// TIA Portal V20 export
DATA_BLOCK "ControlNodes"   // DB72
// stored: MemoryReserve 100, Namespace Unit1.Em7
   VAR
      em : "LAF_typeEmControlNode";
      emstate { S7_SetPoint := 'True'} : "LUC_typeStates";
      cm : "Unit1.Em7.typeCmControlNode";
      citiMap : Struct
         PMC : "LER_PMC_Input_Data";
         FlexNet { S7_SetPoint := 'True'} : "LER_FlexNet_Data";
      END_STRUCT;
      hotPressRight : "Unit1.Em7.typeSequenceControlNode";
      emData : "Unit1.Em7.typeEmDataControlNode";
      SpecialFunctionMode : Struct
         DryRun : Struct
            JRdetectPV : Array[0..15] of Bool;
         END_STRUCT;
      END_STRUCT;
      cmHotPressRightSafetyPin : "LBC_typeDigitalSignalControlNode";
      cmHotPressRightJRDetect : "LBC_typeDigitalSignalControlNode";
      cmHotPressRightStageLiftFrontUpDown : "LBC_typeTwoWayActuatorControlNode";
      cmHotPressRightStageLiftRearUpDown : "LBC_typeTwoWayActuatorControlNode";
      cmHotPressRightStageLiftAllUpDown : "LBC_typeTwoWayActuatorControlNode";
      cmHotPressRightServoPress : "LER_typeServoPressControlNode";
      cmHotPressRightTemperature : "LER_typeHeaterControlNode";
   END_VAR
BEGIN
END_DATA_BLOCK
